// TIA Portal project "AutoCrib" (V16)

(* hardware
DEVICE "S7-1200 station_1"  S7-1200 Station
   slot 0: "Rack_0"  S7-1200 Rack  Rack  V1.0
   slot 1: "PLC_1"  CPU 1214C DC/DC/DC  6ES7 214-1AG40-0XB0  V4.4
   slot 3: "DI 2/DQ 2x24VDC_1"  DI2/DQ2 signal board  6ES7 223-0BD30-0XB0  V1.0
*)

// ===== PLC "PLC_1"  CPU 1214C DC/DC/DC =====

ORGANIZATION_BLOCK "Main"   // OB1, LAD, ProgramCycle
TITLE = "Main Program Sweep (Cycle)"
{ S7_Optimized_Access := 'TRUE' }
VERSION : 0.1
   VAR_INPUT
      Initial_Call : Bool;   // Initial call of this OB
      Remanence : Bool;   // =True, if remanent data are available
   END_VAR
BEGIN

REGION Network 1
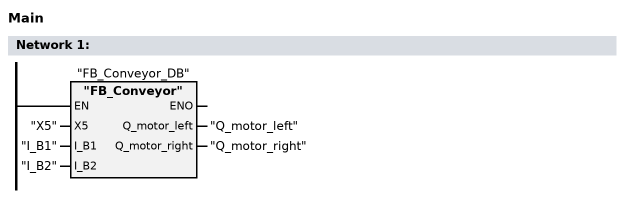
   RUNG wire#powerrail
      "FB_Conveyor_DB"(X5 := "X5", I_B1 := "I_B1", I_B2 := "I_B2", Q_motor_left => "Q_motor_left", Q_motor_right => "Q_motor_right")
   END_RUNG
   // the same network as SCL:
   "FB_Conveyor_DB"(X5 := "X5",   // "FB_Conveyor"
                    I_B1 := "I_B1",
                    I_B2 := "I_B2",
                    Q_motor_left => "Q_motor_left",
                    Q_motor_right => "Q_motor_right");
END_REGION
END_ORGANIZATION_BLOCK